PROGRAM P_Demo_FB_HVACAnalogInput
VAR
    fb : FB_HVACAnalogInput;                            // 被演示 FB 实例
    eDataSecurityType_in : E_HVACDataSecurityType ;
    bSetDefault_in : BOOL := FALSE;
    iRawValue_in : INT := 0;
    tTaskCycleTime_in : TIME := T#0S;
    tCtrlCycleTime_in : TIME := T#0S;
    bEnableLimitCtrl_in : BOOL := FALSE;
    bCtrlVoltage_in : BOOL := FALSE;
    bReset_in : BOOL := FALSE;
    iHighRange_io : INT := 0;
    iLowRange_io : INT := 0;
    rHighRange_io : REAL := 0.0;
    rLowRange_io : REAL := 0.0;
    rHighLimit_io : REAL := 0.0;
    rLowLimit_io : REAL := 0.0;
    tFilterTime_io : TIME := T#0S;
    rOffset_io : REAL := 0.0;
    rPresentValue_out : REAL;
    byState_out : BYTE;
    bError_out : BOOL;
    eErrorCode_out : E_HVACErrorCodes;
    bErrorHighLimit_out : BOOL;
    bErrorLowLimit_out : BOOL;
    bErrorGeneral_out : BOOL;
    byError_out : BYTE;
    bInvalidParameter_out : BOOL;
END_VAR

// ============================================================================
// Tc2_HVAC.FB_HVACAnalogInput 演示程序
// ============================================================================
// 场景：把本 FB 实例化到一个 PLC 程序里，每周期单次调用；按需要把 VAR_INPUT 与
//       VAR_IN_OUT 接到工程信号；VAR_OUTPUT 写入对应监视变量。
// 价值：使用本 FB 比手写状态机 / 控制算法节省大量代码；与 Tc2_HVAC 体系内其它 FB
//       直接对接，命名 / 持久化 / 模式仲裁等约定一致。具体语义见 FB_HVACAnalogInput.md 主文档。
// 验证步骤：
//   1. 右键 PLC 项目下 POUs 文件夹 → Add → Existing Item → 选本 .TcPOU 文件
//   2. 引用 Tc2_HVAC（References → Add library）
//   3. 编译 → 登录 → 运行
//   4. 在线写各 *_in 输入信号触发 FB；在线 monitor *_out 引脚观察状态
// ============================================================================

fb(
    eDataSecurityType := eDataSecurityType_in,
    bSetDefault := bSetDefault_in,
    iRawValue := iRawValue_in,
    tTaskCycleTime := tTaskCycleTime_in,
    tCtrlCycleTime := tCtrlCycleTime_in,
    bEnableLimitCtrl := bEnableLimitCtrl_in,
    bCtrlVoltage := bCtrlVoltage_in,
    bReset := bReset_in,
    iHighRange := iHighRange_io,
    iLowRange := iLowRange_io,
    rHighRange := rHighRange_io,
    rLowRange := rLowRange_io,
    rHighLimit := rHighLimit_io,
    rLowLimit := rLowLimit_io,
    tFilterTime := tFilterTime_io,
    rOffset := rOffset_io,
    rPresentValue => rPresentValue_out,
    byState => byState_out,
    bError => bError_out,
    eErrorCode => eErrorCode_out,
    bErrorHighLimit => bErrorHighLimit_out,
    bErrorLowLimit => bErrorLowLimit_out,
    bErrorGeneral => bErrorGeneral_out,
    byError => byError_out,
    bInvalidParameter => bInvalidParameter_out
);

END_PROGRAM

(* stored: Version 1.1.0.1, ProductVersion 3.1.4024.5
   POU P_Demo_FB_HVACAnalogInput: Id {d3720ad0-efb7-50c9-a476-9f7f1d6c51b1}, SpecialFunc None *)
